# B&R Automation Studio project TFG2024
Automation Studio 4.12.2.93; technology packages: mappMotion 5.24.1

## Configuration Config1

CPU X20CP0483, AutomationRuntime B4.93, Build 4.1.2, Vc V4.72.6

### Hardware
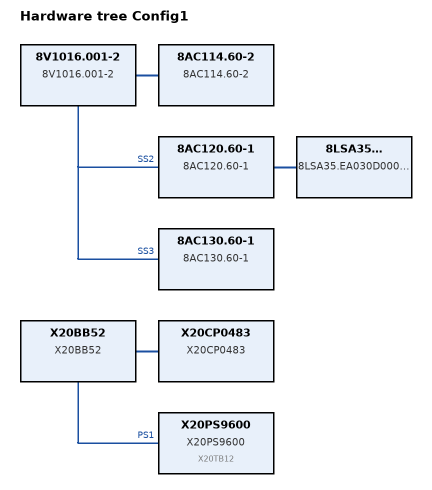
```
8AC114.60-2 : 8AC114.60-2 v1.0.0.8  [SS -> 8V1016.001-2.SS1; PLK1 -> X20CP0483.IF3 (NodeNumber=1) [Cable Type=PowerlinkCable, Length=10, Version=1.0.0.3]]
8AC120.60-1 : 8AC120.60-1 v2.2.0.0  [SS -> 8V1016.001-2.SS2]
  PlugInType = Encoder
  McAcoposTypeID = AcoposPlugInConfig
8AC130.60-1 : 8AC130.60-1 v2.2.0.0  [SS -> 8V1016.001-2.SS3]
8LSA35.EA030D000-0 : 8LSA35.EA030D000-0 v1.0.4.40  [EC -> 8AC120.60-1.EC; MT -> 8V1016.001-2.MT1]
8V1016.001-2 : 8V1016.001-2 v2.2.0.0
  DriveConfiguration/Module:
    McAcoposTypeID = AcoposConfig
    ActivateACOPOSSimulationOnPLC = 1
  DriveConfiguration/Channel[1]/RealAxis:
    AxisReference = gAxis_1
    MechanicalElementsIsInvisible = 0
  DriveConfiguration/Channel[1]/RealAxis/MechanicalElements/Gearbox:
    InputIsReadOnly = 0
    Input = 1
    OutputIsReadOnly = 0
    Output = 1
  DriveConfiguration/Channel[1]/RealAxis/MechanicalElements/RotaryToLinearTransformation:
    ReferenceDistanceIsReadOnly = 0
    ReferenceDistance = 1
  DriveConfiguration/Channel[1]/RealAxis/Controller:
    ModeIsReadOnly = 0
    Mode = PositionController
  DriveConfiguration/Channel[1]/RealAxis/Controller/Mode/Position:
    ProportionalGain = 50.0
    IntegrationTime = 0.0
    PredictionTime = 0.0004
    TotalDelayTime = 0.0004
  DriveConfiguration/Channel[1]/RealAxis/Controller/Mode/Speed:
    ProportionalGainIsReadOnly = 0
    ProportionalGain = 2.0
    IntegrationTimeIsReadOnly = 0
    IntegrationTime = 0.0
    FilterTimeIsReadOnly = 0
    FilterTime = 0.0
  DriveConfiguration/Channel[1]/RealAxis/Controller/Mode/LoopFilters:
    LoopFilterXIsReadOnly = 0
    LoopFilter1 = NotUsed
    LoopFilter2 = NotUsed
    LoopFilter3 = NotUsed
  DriveConfiguration/Channel[1]/RealAxis/Homing:
    ModeIsReadOnly = 0
    Mode = Direct
  DriveConfiguration/Channel[1]/RealAxis/Homing/Mode:
    Position = 0.0
    ReferencePulse = NotUsed
  DriveConfiguration/Channel[1]/RealAxis/Homing:
    RestorePositionVariable = 
  DriveConfiguration/Channel[1]/RealAxis/StopReaction:
    QuickstopIsReadOnly = 0
    Quickstop = DecelerationLimit
    DriveErrorIsReadOnly = 0
    DriveError = DecelerationLimit
  DriveConfiguration/Channel[1]/RealAxis/MovementErrorLimits:
    PositionError = 1.0
    VelocityErrorMonitoring = Automatic1
  DriveConfiguration/Channel[1]/RealAxis:
    JerkFilterIsReadOnly = 0
    JerkFilter = NotUsed
    ZeroVibrationFilter = NotUsed
  DriveConfiguration/Channel[1]/RealAxis/DigitalInputs/HomingSwitch:
    SourceIsReadOnly = 0
    Source = X1Ref
    Level = High
  DriveConfiguration/Channel[1]/RealAxis/DigitalInputs/PositiveLimitSwitch:
    Source = X1PosLim
    Level = High
  DriveConfiguration/Channel[1]/RealAxis/DigitalInputs/NegativeLimitSwitch:
    Source = X1NegLim
    Level = High
  DriveConfiguration/Channel[1]/RealAxis/DigitalInputs/Trigger1:
    Source = X1Trigger1
    Level = High
  DriveConfiguration/Channel[1]/RealAxis/DigitalInputs/Trigger2:
    Source = X1Trigger2
    Level = High
  DriveConfiguration/Channel[1]/RealAxis/DigitalInputs/Quickstop:
    Input = Trigger2
  DriveConfiguration/Channel[1]/RealAxis/Simulation:
    SimulationModeOnPLC = SetValueGeneration
    SimulationModeOnACOPOS = NotUsed
  DriveConfiguration/Channel[1]:
    ExternalEncoderAxis = NotUsed
X20BB52 : X20BB52 v1.2.0.0
X20CP0483 : X20CP0483 v1.6.0.0  [SL -> X20BB52.SL1]
  Connector IF2:
    ActivateDevice = 1
  Connector IF3:
    ActivateANSL = 1
  ConfigurationID = TFG2024_Config1
  Simulation = 1
  TimerDeviceType = SWIOTIMER
  Cyclic1Duration = 10000
  Cyclic1Tolerance = 10000
  Cyclic2Duration = 20000
  Cyclic2Tolerance = 20000
  Cyclic3Duration = 50000
  Cyclic3Tolerance = 50000
  Cyclic4Duration = 100000
  Cyclic4Tolerance = 100000
  Cyclic5Duration = 200000
  Cyclic5Tolerance = 200000
  Cyclic6Duration = 500000
  Cyclic6Tolerance = 500000
  Cyclic7Duration = 1000000
  Cyclic7Tolerance = 1000000
  Cyclic8Duration = 10000
  Cyclic8Tolerance = 30000000
  FileDevice1
  FileDeviceName1 = USER
  FileDevicePath1 = USER_PATH
  ActivateOpcUa = 1
  OpcUaInformationModels_PV_Version = 1
X20PS9600 : X20PS9600 v1.6.0.0  [PS -> X20BB52.PS1; SS1 -> X20TB12.SS]
X20TB12 : X20TB12 v1.0.0.0
```

### AxisConfig.axis - X20CP0483/mappMotion/AxisConfig.axis
```
Element gAxis_1 (Type=axis)
  BaseTypeIsReadOnly = 0
  BaseType = RotaryPeriodic
    MeasurementUnitIsReadOnly = 0
    MeasurementUnit = 17476
    MeasurementResolutionIsReadOnly = 0
    MeasurementResolution = 0.001
    CountDirectionIsReadOnly = 0
    CountDirection = Standard
    PeriodSettings:
      Period = 360.0
  MovementLimitsIsReadOnly = 0
  MovementLimits = Internal
    Position:
      LowerLimitMin = -1.79769313486231E308
      UpperLimitMax = 1.79769313486231E308
      LowerLimit = -1000.0
      UpperLimit = 1000.0
    VelocityIsReadOnly = 0
    Velocity:
      VelocityMax = 3.4E38
      Velocity = 3600
    AccelerationIsReadOnly = 0
    Acceleration:
      AccelerationMax = 3.4E38
      Acceleration = 36000
    DecelerationIsReadOnly = 0
    Deceleration:
      DecelerationMax = 3.4E38
      Deceleration = 36000
  Alarms = None
```

## Logical view

### Global.typ - Global data types
```iecst
TYPE
	Alarm : 	STRUCT
		Status : BOOL;
		Description : WSTRING[80];
		Severity : USINT;
		Acknowledgement : BOOL;
	END_STRUCT;
END_TYPE
```

### Global.var - Global variables
```iecst
VAR
	MpAxisBasic_0 : MpAxisBasic;
	AxisParam : MpAxisBasicParType;

	Alarm1 : Alarm;

END_VAR
```

### Program Logical/Axis1Ctrl (IEC)

#### Cyclic.ld
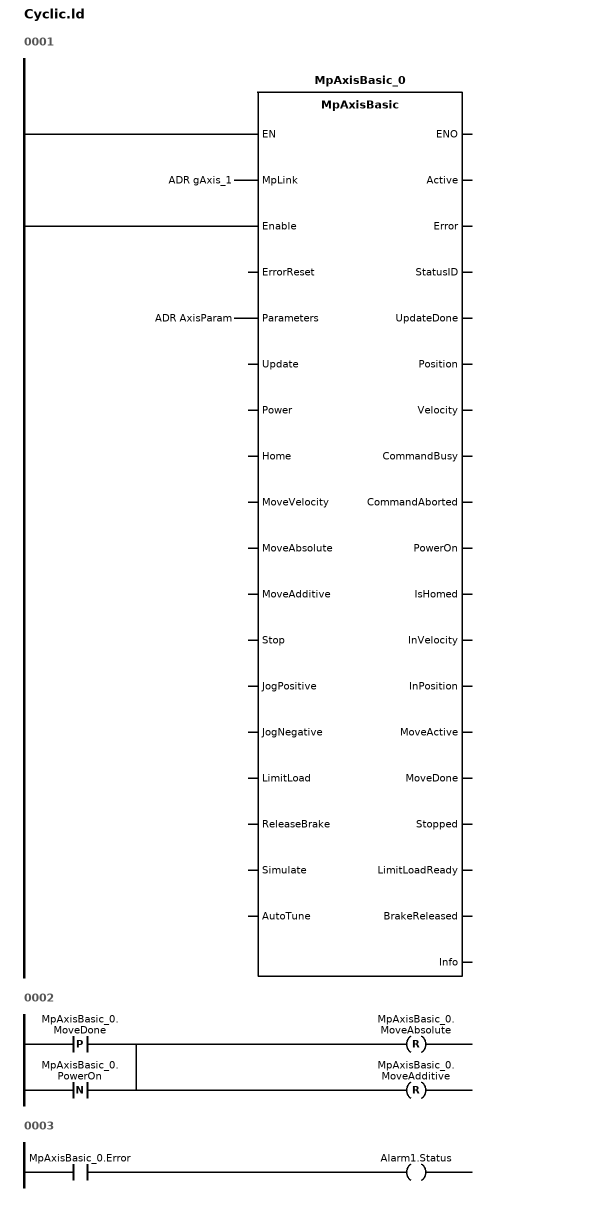
Ladder, written as Structured Text:
```iecst
PROGRAM _CYCLIC
VAR
    _e1 : R_TRIG;
    _e2 : F_TRIG;
END_VAR
(* Network 1 *)
MpAxisBasic_0(MpLink := ADR(gAxis_1), Enable := TRUE, Parameters := ADR(AxisParam));

(* Network 2 *)
_e1(CLK := MpAxisBasic_0.MoveDone);
_e2(CLK := MpAxisBasic_0.PowerOn);
IF _e1.Q OR _e2.Q THEN
    MpAxisBasic_0.MoveAbsolute := FALSE;
    MpAxisBasic_0.MoveAdditive := FALSE;
END_IF;

(* Network 3 *)
Alarm1.Status := MpAxisBasic_0.Error;
END_PROGRAM
```

#### Exit.ld
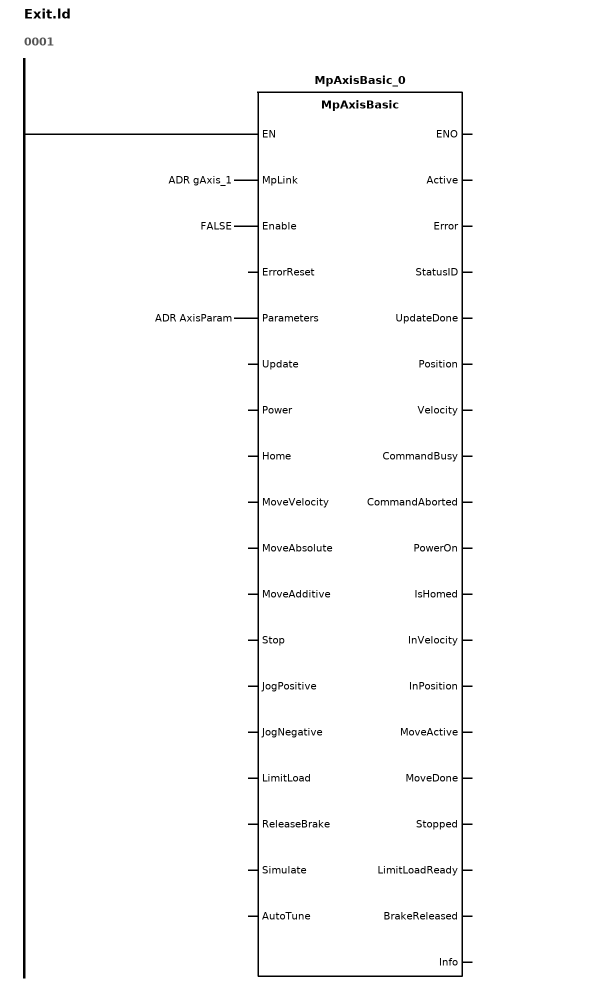
Ladder, written as Structured Text:
```iecst
PROGRAM _EXIT
(* Network 1 *)
MpAxisBasic_0(MpLink := ADR(gAxis_1), Enable := FALSE, Parameters := ADR(AxisParam));
END_PROGRAM
```

#### Init.ld
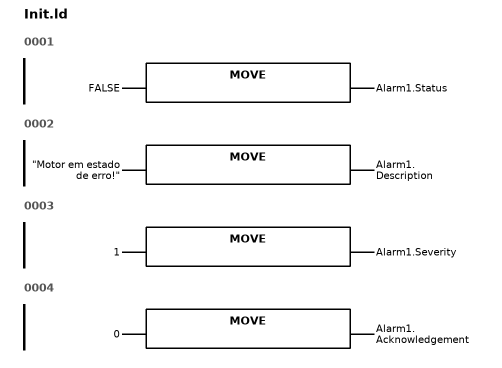
Ladder, written as Structured Text:
```iecst
PROGRAM _INIT
(* Network 1 *)
Alarm1.Status := FALSE;

(* Network 2 *)
Alarm1.Description := "Motor em estado de erro!";

(* Network 3 *)
Alarm1.Severity := 1;

(* Network 4 *)
Alarm1.Acknowledgement := 0;
END_PROGRAM
```

Listed in the project but not available here: Logical/Libraries
